// TIA Portal V19 export
TYPE "LAF_typeXyzhandlingEm4ParametersInterfaceHmi"
// stored: Access Published
   STRUCT
      configuration : "LAF_typeXyzhandlingEm4ParametersHmi";
      commands : "LBC_typeInterfaceCommands";
      monitoring { S7_SetPoint := 'True'} : "LAF_typeXyzhandlingEm4ProcessValuesHmi";
   END_STRUCT;
END_TYPE
